TYPE T_AVL_Node : ST_AVL_NODE; END_TYPE

(* stored: Version 1.1.0.1, ProductVersion 3.1.4024.4
   DUT T_AVL_Node: Id {d8cc1851-ba66-4b92-881d-7cda2a0f3dd9} *)
